// TIA Portal V20 export
TYPE "typeSafetySensor"
// stored: Access Published, IsFailsafeCompliant true, Namespace Safety
   STRUCT
      anodeCvCoverBwd : Bool;   // Anode Conveyor Cover Backward
      cathodeCvCoverBwd : Bool;   // Cathode Conveyor Cover Backward
      anodeCvCoverFwd : Bool;   // Anode Conveyor Cover Forward
      cathodeCvCoverFwd : Bool;   // Cathode Conveyor Cover Forward
   END_STRUCT;
END_TYPE
